FUNCTION_BLOCK ALI_FB_CTUD (* Up-Down counter (LINT) ALI-Adapter Version *)
  (* Standard: 61499-2; Description: Copyright (c) 2026 Meisterschulen am Ostbahnhof This program and the accompanying materials are made available under the terms of the Eclipse Public License 2.0 which is available at https://www.eclipse.org/legal/epl-2.0/ SPDX-License-Identifier: EPL-2.0 NOTE: This block fires the AX output events (QU.E1, QD.E1) on every update (CU, CD, R, LD, PV). If on-change triggering is required, use of an AX_D_FF as a filter is recommended. *)
  (* Version 1.0, 2026-04-21, Franz Höpfinger, Meisterschulen am Ostbahnhof, initial API and implementation and/or initial documentation *)
  PACKAGE adapter::iec61131_3::counters;
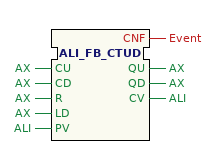
  EVENT_OUTPUT
    CNF; (* Execution Confirmation *)
  END_EVENT
  SOCKETS
    CU : adapter::types::unidirectional::AX; (* Count up *)
    CD : adapter::types::unidirectional::AX; (* Count down *)
    R : adapter::types::unidirectional::AX; (* Reset *)
    LD : adapter::types::unidirectional::AX; (* Load *)
    PV : adapter::types::unidirectional::ALI; (* Preset value *)
  END_SOCKETS
  PLUGS
    QU : adapter::types::unidirectional::AX; (* Output Up *)
    QD : adapter::types::unidirectional::AX; (* Output Down *)
    CV : adapter::types::unidirectional::ALI; (* Count value *)
  END_PLUGS
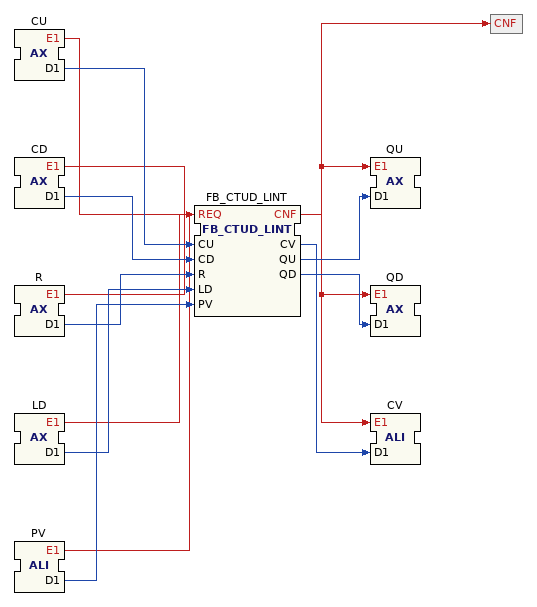
  FBS
    FB_CTUD_LINT : iec61131::counters::FB_CTUD_LINT;
  END_FBS
  EVENT_CONNECTIONS
    CU.E1 TO FB_CTUD_LINT.REQ;
    CD.E1 TO FB_CTUD_LINT.REQ;
    R.E1 TO FB_CTUD_LINT.REQ;
    LD.E1 TO FB_CTUD_LINT.REQ;
    PV.E1 TO FB_CTUD_LINT.REQ;
    FB_CTUD_LINT.CNF TO CV.E1;
    FB_CTUD_LINT.CNF TO QU.E1;
    FB_CTUD_LINT.CNF TO QD.E1;
    FB_CTUD_LINT.CNF TO CNF;
  END_CONNECTIONS
  DATA_CONNECTIONS
    CU.D1 TO FB_CTUD_LINT.CU;
    CD.D1 TO FB_CTUD_LINT.CD;
    R.D1 TO FB_CTUD_LINT.R;
    LD.D1 TO FB_CTUD_LINT.LD;
    PV.D1 TO FB_CTUD_LINT.PV;
    FB_CTUD_LINT.CV TO CV.D1;
    FB_CTUD_LINT.QU TO QU.D1;
    FB_CTUD_LINT.QD TO QD.D1;
  END_CONNECTIONS
END_FUNCTION_BLOCK
